{attribute 'qualified_only'}
{attribute 'strict'}
TYPE eExternalControlMode :
(
	off := 0,
	Readonly := 1,
	BasicControl := 2,
	AdvancedControl := 3
);
END_TYPE

(* stored: Version 1.1.0.1, ProductVersion 3.1.4024.12
   DUT eExternalControlMode: Id {f6dd61a0-169c-4719-8409-3ddb1d74c7c0} *)
